// This function has been automatically generated from the project information.
{attribute 'signature_flag' := '1073741824'}
{attribute 'TcGenerated'}
{attribute 'no-analysis'}
FUNCTION F_GetTitle : WSTRING
VAR_INPUT
	
END_VAR

F_GetTitle := "Library_OOP_Course";

END_FUNCTION

(* stored: Version 1.1.0.1
   POU F_GetTitle: Id {cf1d2fa5-4562-0076-0554-34ee66c96922}, SpecialFunc None *)
